(* Logix 5000 project; controller NSH_PLC2 vendor 1 type 14 code 167 rev 32.14; software revision 32.03; part 3 of 6 *)
(* tags used below, declared in another part *)
   AOI_MCC2_15J_ToPLC1 : E300ToMotor;
   AOI_MCC2_15L_ToPLC1 : E300ToMotor;
   AOI_MCC2_16A_ToPLC1 : E300ToMotor;
   AOI_MCC2_16C_ToPLC1 : E300ToMotor;
   AOI_MCC2_16E_ToPLC1 : E300ToMotor;
   AOI_MCC2_16G_ToPLC1 : E300ToMotor;
   AOI_MCC2_16J_ToPLC1 : E300ToMotor;
   AOI_MCC2_16L_ToPLC1 : E300ToMotor;
   AOI_MCC2_17A_ToPLC1 : E300ToMotor;
   AOI_MCC2_17C_ToPLC1 : E300ToMotor;
   AOI_MCC2_17E_ToPLC1 : E300ToMotor;
   AOI_MCC2_17G_ToPLC1 : E300ToMotor;
   AOI_MCC2_17J_ToPLC1 : E300ToMotor;
   AOI_MCC2_18A_ToPLC1 : E300ToMotor;
   AOI_MCC2_18C_ToPLC1 : E300ToMotor;
   AOI_MCC2_18E_ToPLC1 : E300ToMotor;
   AOI_MCC2_18G_ToPLC1 : E300ToMotor;
   AOI_MCC2_18J_ToPLC1 : E300ToMotor;
   AOI_MCC2_18L_ToPLC1 : E300ToMotor;
   AOI_MCC2_19A_ToPLC1 : E300ToMotor;
   AOI_MCC2_19C_ToPLC1 : E300ToMotor;
   AOI_MCC2_19E_ToPLC1 : E300ToMotor;
   AOI_MCC2_19G_ToPLC1 : E300ToMotor;
   AOI_MCC2_19J_ToPLC1 : E300ToMotor;
   AOI_MCC2_19L_ToPLC1 : E300ToMotor;
   AOI_MCC2_20C_ToPLC1 : E300ToMotor;
   AOI_MCC2_20E_ToPLC1 : E300ToMotor;
   AOI_MCC2_20G_ToPLC1 : E300ToMotor;
   AOI_MCC2_20J_ToPLC1 : E300ToMotor;
   AOI_MCC2_21A_ToPLC1 : E300ToMotor;
   AOI_MCC2_21C_ToPLC1 : E300ToMotor;
   AOI_MCC2_21E_ToPLC1 : E300ToMotor;
   AOI_MCC2_21G_ToPLC1 : PF525ToMotor;
   AOI_MCC2_21K_ToPLC1 : PF525ToMotor;
   AOI_MCC3_10A_ToPLC1 : E300ToMotor;
   AOI_MCC3_10D_ToPLC1 : E300ToMotor;
   AOI_MCC3_10G_ToPLC1 : E300ToMotor;
   AOI_MCC3_2A_ToPLC1 : PF525ToMotor;
   AOI_MCC3_2D_ToPLC1 : PF525ToMotor;
   AOI_MCC3_2G_ToPLC1 : PF525ToMotor;
   AOI_MCC3_2K_ToPLC1 : PF525ToMotor;
   AOI_MCC3_3A_ToPLC1 : PF525ToMotor;
   AOI_MCC3_3D_ToPLC1 : PF525ToMotor;
   AOI_MCC3_3G_ToPLC1 : PF525ToMotor;
   AOI_MCC3_3K_ToPLC1 : PF525ToMotor;
   AOI_MCC3_4A_ToPLC1 : PF525ToMotor;
   AOI_MCC3_4D_ToPLC1 : PF525ToMotor;
   AOI_MCC3_4G_ToPLC1 : PF525ToMotor;
   AOI_MCC3_4K_ToPLC1 : PF525ToMotor;
   AOI_MCC3_5A_ToPLC1 : PF525ToMotor;
   AOI_MCC3_5D_ToPLC1 : PF525ToMotor;
   AOI_MCC3_5G_ToPLC1 : PF525ToMotor;
   AOI_MCC3_5K_ToPLC1 : PF525ToMotor;
   AOI_MCC3_6A_ToPLC1 : PF525ToMotor;
   AOI_MCC3_6D_ToPLC1 : PF525ToMotor;
   AOI_MCC3_6G_ToPLC1 : E300ToMotor;
   AOI_MCC3_6J_ToPLC1 : E300ToMotor;
   AOI_MCC3_7A_ToPLC1 : E300ToMotor;
   AOI_MCC3_7C_ToPLC1 : E300ToMotor;
   AOI_MCC3_7E_ToPLC1 : E300ToMotor;
   AOI_MCC3_7G_ToPLC1 : PF525ToMotor;
   AOI_MCC3_7K_ToPLC1 : PF525ToMotor;
   AOI_MCC3_8A_ToPLC1 : E300ToMotor;
   AOI_MCC3_8D_ToPLC1 : PF525ToMotor;
   AOI_MCC3_8H_ToPLC1 : E300ToMotor;
   AOI_MCC3_8K_ToPLC1 : PF525ToMotor;
   AOI_MCC3_9A_ToPLC1 : E300ToMotor;
   AOI_MCC3_9C_ToPLC1 : E300ToMotor;
   AOI_MCC3_9E_ToPLC1 : E300ToMotor;
   AOI_MCC3_9G_ToPLC1 : E300ToMotor;
   AOI_MCC3_9J_ToPLC1 : E300ToMotor;
   AOI_MCC3_9L_ToPLC1 : E300ToMotor;
   Const_4000_Hex : INT;   // Constant #16:4000, Entry Status Communicating
   GSV_EntryStatus : INT;   // GSV Entry Status, shold be #16:4000
   MCC2_15J_CommsOK : BOOL;   // Communications with AOP OK
   MCC2_15L_CommsOK : BOOL;   // Communications with AOP OK
   MCC2_16A_CommsOK : BOOL;   // Communications with AOP OK
   MCC2_16C_CommsOK : BOOL;   // Communications with AOP OK
   MCC2_16E_CommsOK : BOOL;   // Communications with AOP OK
   MCC2_16G_CommsOK : BOOL;   // Communications with AOP OK
   MCC2_16J_CommsOK : BOOL;   // Communications with AOP OK
   MCC2_16L_CommsOK : BOOL;   // Communications with AOP OK
   MCC2_17A_CommsOK : BOOL;   // Communications with AOP OK
   MCC2_17C_CommsOK : BOOL;   // Communications with AOP OK
   MCC2_17E_CommsOK : BOOL;   // Communications with AOP OK
   MCC2_17G_CommsOK : BOOL;   // Communications with AOP OK
   MCC2_17J_CommsOK : BOOL;   // Communications with AOP OK
   MCC2_18A_CommsOK : BOOL;   // Communications with AOP OK
   MCC2_18C_CommsOK : BOOL;   // Communications with AOP OK
   MCC2_18E_CommsOK : BOOL;   // Communications with AOP OK
   MCC2_18G_CommsOK : BOOL;   // Communications with AOP OK
   MCC2_18J_CommsOK : BOOL;   // Communications with AOP OK
   MCC2_18L_CommsOK : BOOL;   // Communications with AOP OK
   MCC2_19A_CommsOK : BOOL;   // Communications with AOP OK
   MCC2_19C_CommsOK : BOOL;   // Communications with AOP OK
   MCC2_19E_CommsOK : BOOL;   // Communications with AOP OK
   MCC2_19G_CommsOK : BOOL;   // Communications with AOP OK
   MCC2_19J_CommsOK : BOOL;   // Communications with AOP OK
   MCC2_19L_CommsOK : BOOL;   // Communications with AOP OK
   MCC2_20C_CommsOK : BOOL;   // Communications with AOP OK
   MCC2_20E_CommsOK : BOOL;   // Communications with AOP OK
   MCC2_20G_CommsOK : BOOL;   // Communications with AOP OK
   MCC2_20J_CommsOK : BOOL;   // Communications with AOP OK
   MCC2_21A_CommsOK : BOOL;   // Communications with AOP OK
   MCC2_21C_CommsOK : BOOL;   // Communications with AOP OK
   MCC2_21E_CommsOK : BOOL;   // Communications with AOP OK
   MCC2_21G_CommsOK : BOOL;   // Communications with AOP OK
   MCC2_21K_CommsOK : BOOL;   // Communications with AOP OK
   MCC3_10A_CommsOK : BOOL;   // Communications with AOP OK
   MCC3_10D_CommsOK : BOOL;   // Communications with AOP OK
   MCC3_10G_CommsOK : BOOL;   // Communications with AOP OK
   MCC3_2A_CommsOK : BOOL;   // Communications with AOP OK
   MCC3_2D_CommsOK : BOOL;   // Communications with AOP OK
   MCC3_2G_CommsOK : BOOL;   // Communications with AOP OK
   MCC3_2K_CommsOK : BOOL;   // Communications with AOP OK
   MCC3_3A_CommsOK : BOOL;   // Communications with AOP OK
   MCC3_3D_CommsOK : BOOL;   // Communications with AOP OK
   MCC3_3G_CommsOK : BOOL;   // Communications with AOP OK
   MCC3_3K_CommsOK : BOOL;   // Communications with AOP OK
   MCC3_4A_CommsOK : BOOL;   // Communications with AOP OK
   MCC3_4D_CommsOK : BOOL;   // Communications with AOP OK
   MCC3_4G_CommsOK : BOOL;   // Communications with AOP OK
   MCC3_4K_CommsOK : BOOL;   // Communications with AOP OK
   MCC3_5A_CommsOK : BOOL;   // Communications with AOP OK
   MCC3_5D_CommsOK : BOOL;   // Communications with AOP OK
   MCC3_5G_CommsOK : BOOL;   // Communications with AOP OK
   MCC3_5K_CommsOK : BOOL;   // Communications with AOP OK
   MCC3_6A_CommsOK : BOOL;   // Communications with AOP OK
   MCC3_6D_CommsOK : BOOL;   // Communications with AOP OK
   MCC3_6G_CommsOK : BOOL;   // Communications with AOP OK
   MCC3_6J_CommsOK : BOOL;   // Communications with AOP OK
   MCC3_7A_CommsOK : BOOL;   // Communications with AOP OK
   MCC3_7C_CommsOK : BOOL;   // Communications with AOP OK
   MCC3_7E_CommsOK : BOOL;   // Communications with AOP OK
   MCC3_7G_CommsOK : BOOL;   // Communications with AOP OK
   MCC3_7K_CommsOK : BOOL;   // Communications with AOP OK
   MCC3_8A_CommsOK : BOOL;   // Communications with AOP OK
   MCC3_8D_CommsOK : BOOL;   // Communications with AOP OK
   MCC3_8H_CommsOK : BOOL;   // Communications with AOP OK
   MCC3_8K_CommsOK : BOOL;   // Communications with AOP OK
   MCC3_9A_CommsOK : BOOL;   // Communications with AOP OK
   MCC3_9C_CommsOK : BOOL;   // Communications with AOP OK
   MCC3_9E_CommsOK : BOOL;   // Communications with AOP OK
   MCC3_9G_CommsOK : BOOL;   // Communications with AOP OK
   MCC3_9J_CommsOK : BOOL;   // Communications with AOP OK
   MCC3_9L_CommsOK : BOOL;   // Communications with AOP OK
   MotorsStatusTag : MotorsStatusUDT;   // Only Instance of UDT
(* MainProgram, continued *)

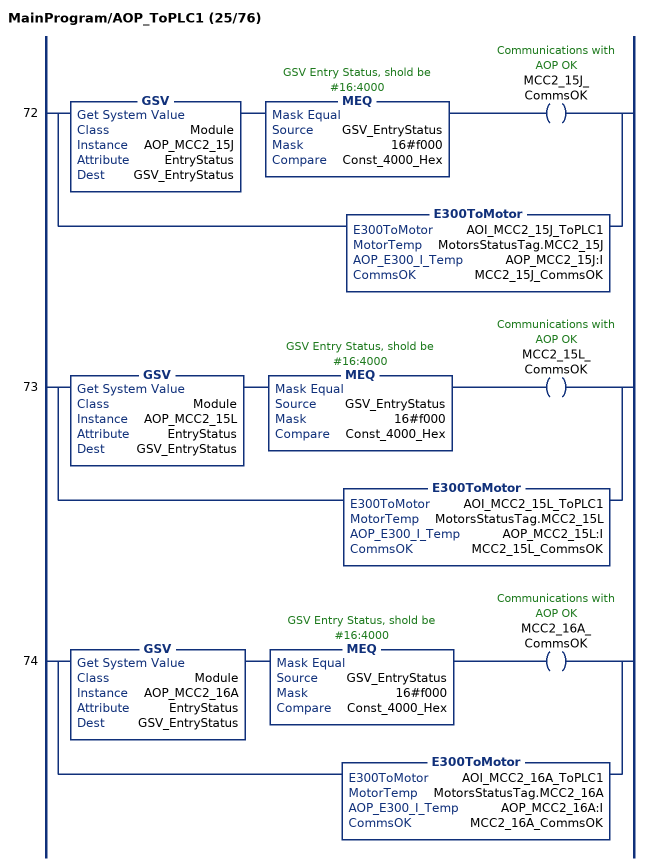
   [picture p31: MainProgram/AOP_ToPLC1 rungs 72-74]
   72: [GSV(Module,AOP_MCC2_15J,EntryStatus,GSV_EntryStatus) MEQ(GSV_EntryStatus,16#f000,Const_4000_Hex) OTE(MCC2_15J_CommsOK) ,E300ToMotor(AOI_MCC2_15J_ToPLC1,MotorsStatusTag.MCC2_15J,AOP_MCC2_15J:I,MCC2_15J_CommsOK) ];
   73: [GSV(Module,AOP_MCC2_15L,EntryStatus,GSV_EntryStatus) MEQ(GSV_EntryStatus,16#f000,Const_4000_Hex) OTE(MCC2_15L_CommsOK) ,E300ToMotor(AOI_MCC2_15L_ToPLC1,MotorsStatusTag.MCC2_15L,AOP_MCC2_15L:I,MCC2_15L_CommsOK) ];
   74: [GSV(Module,AOP_MCC2_16A,EntryStatus,GSV_EntryStatus) MEQ(GSV_EntryStatus,16#f000,Const_4000_Hex) OTE(MCC2_16A_CommsOK) ,E300ToMotor(AOI_MCC2_16A_ToPLC1,MotorsStatusTag.MCC2_16A,AOP_MCC2_16A:I,MCC2_16A_CommsOK) ];
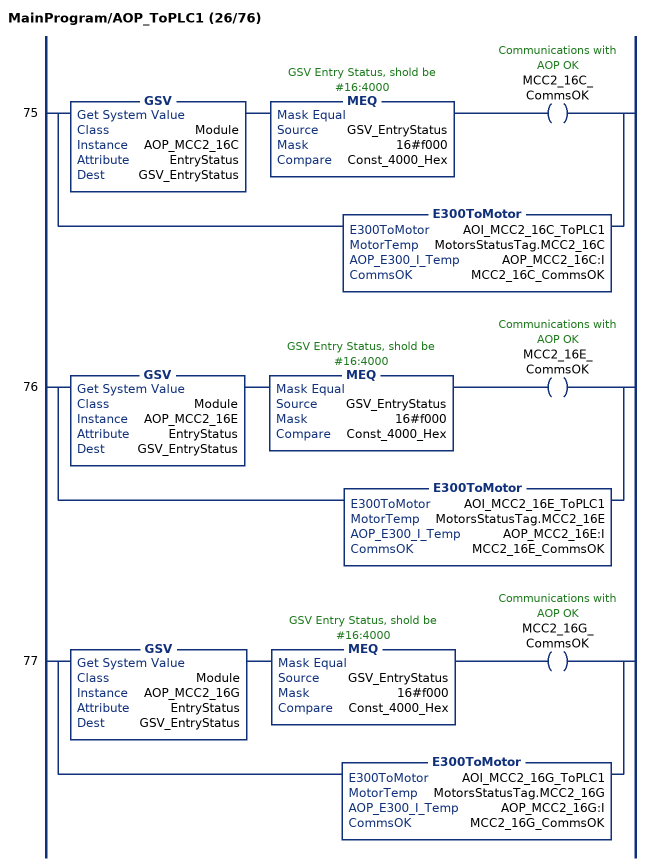
   75: [GSV(Module,AOP_MCC2_16C,EntryStatus,GSV_EntryStatus) MEQ(GSV_EntryStatus,16#f000,Const_4000_Hex) OTE(MCC2_16C_CommsOK) ,E300ToMotor(AOI_MCC2_16C_ToPLC1,MotorsStatusTag.MCC2_16C,AOP_MCC2_16C:I,MCC2_16C_CommsOK) ];
   76: [GSV(Module,AOP_MCC2_16E,EntryStatus,GSV_EntryStatus) MEQ(GSV_EntryStatus,16#f000,Const_4000_Hex) OTE(MCC2_16E_CommsOK) ,E300ToMotor(AOI_MCC2_16E_ToPLC1,MotorsStatusTag.MCC2_16E,AOP_MCC2_16E:I,MCC2_16E_CommsOK) ];
   77: [GSV(Module,AOP_MCC2_16G,EntryStatus,GSV_EntryStatus) MEQ(GSV_EntryStatus,16#f000,Const_4000_Hex) OTE(MCC2_16G_CommsOK) ,E300ToMotor(AOI_MCC2_16G_ToPLC1,MotorsStatusTag.MCC2_16G,AOP_MCC2_16G:I,MCC2_16G_CommsOK) ];
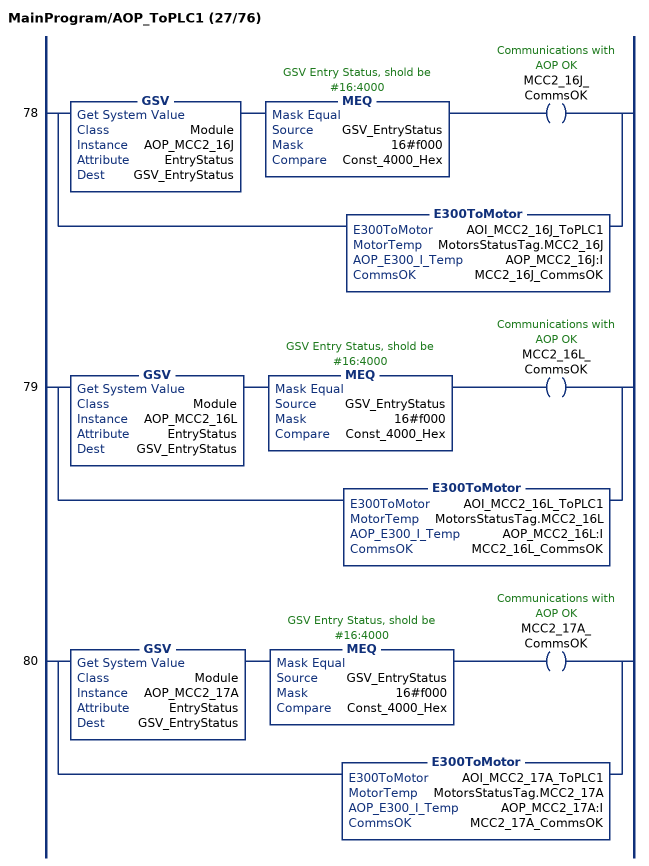
   78: [GSV(Module,AOP_MCC2_16J,EntryStatus,GSV_EntryStatus) MEQ(GSV_EntryStatus,16#f000,Const_4000_Hex) OTE(MCC2_16J_CommsOK) ,E300ToMotor(AOI_MCC2_16J_ToPLC1,MotorsStatusTag.MCC2_16J,AOP_MCC2_16J:I,MCC2_16J_CommsOK) ];
   79: [GSV(Module,AOP_MCC2_16L,EntryStatus,GSV_EntryStatus) MEQ(GSV_EntryStatus,16#f000,Const_4000_Hex) OTE(MCC2_16L_CommsOK) ,E300ToMotor(AOI_MCC2_16L_ToPLC1,MotorsStatusTag.MCC2_16L,AOP_MCC2_16L:I,MCC2_16L_CommsOK) ];
   80: [GSV(Module,AOP_MCC2_17A,EntryStatus,GSV_EntryStatus) MEQ(GSV_EntryStatus,16#f000,Const_4000_Hex) OTE(MCC2_17A_CommsOK) ,E300ToMotor(AOI_MCC2_17A_ToPLC1,MotorsStatusTag.MCC2_17A,AOP_MCC2_17A:I,MCC2_17A_CommsOK) ];
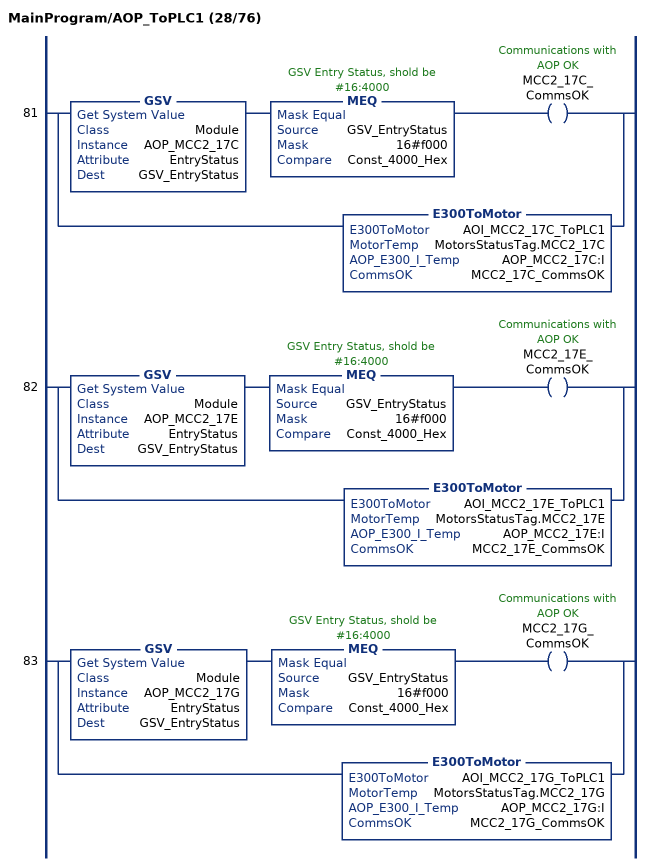
   81: [GSV(Module,AOP_MCC2_17C,EntryStatus,GSV_EntryStatus) MEQ(GSV_EntryStatus,16#f000,Const_4000_Hex) OTE(MCC2_17C_CommsOK) ,E300ToMotor(AOI_MCC2_17C_ToPLC1,MotorsStatusTag.MCC2_17C,AOP_MCC2_17C:I,MCC2_17C_CommsOK) ];
   82: [GSV(Module,AOP_MCC2_17E,EntryStatus,GSV_EntryStatus) MEQ(GSV_EntryStatus,16#f000,Const_4000_Hex) OTE(MCC2_17E_CommsOK) ,E300ToMotor(AOI_MCC2_17E_ToPLC1,MotorsStatusTag.MCC2_17E,AOP_MCC2_17E:I,MCC2_17E_CommsOK) ];
   83: [GSV(Module,AOP_MCC2_17G,EntryStatus,GSV_EntryStatus) MEQ(GSV_EntryStatus,16#f000,Const_4000_Hex) OTE(MCC2_17G_CommsOK) ,E300ToMotor(AOI_MCC2_17G_ToPLC1,MotorsStatusTag.MCC2_17G,AOP_MCC2_17G:I,MCC2_17G_CommsOK) ];
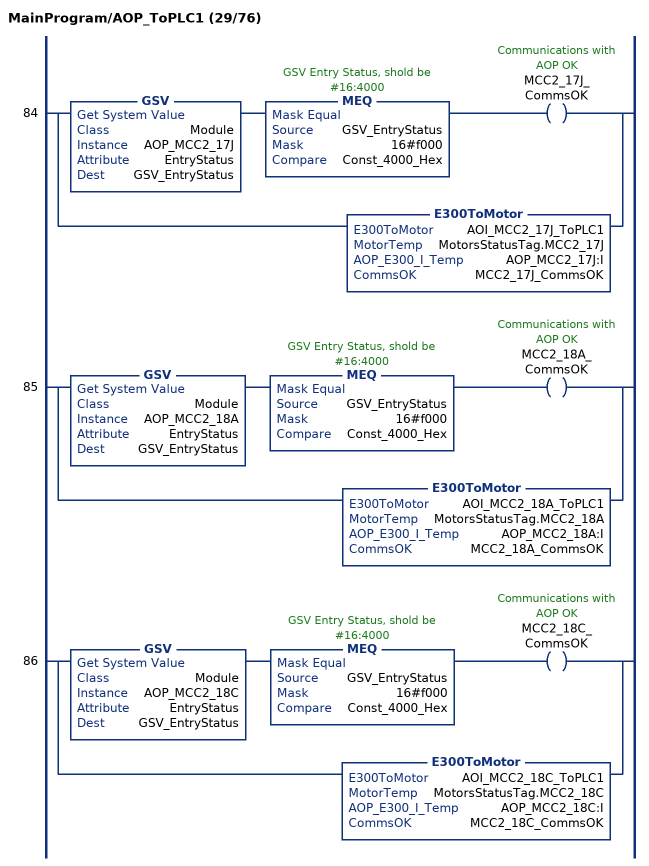
   84: [GSV(Module,AOP_MCC2_17J,EntryStatus,GSV_EntryStatus) MEQ(GSV_EntryStatus,16#f000,Const_4000_Hex) OTE(MCC2_17J_CommsOK) ,E300ToMotor(AOI_MCC2_17J_ToPLC1,MotorsStatusTag.MCC2_17J,AOP_MCC2_17J:I,MCC2_17J_CommsOK) ];
   85: [GSV(Module,AOP_MCC2_18A,EntryStatus,GSV_EntryStatus) MEQ(GSV_EntryStatus,16#f000,Const_4000_Hex) OTE(MCC2_18A_CommsOK) ,E300ToMotor(AOI_MCC2_18A_ToPLC1,MotorsStatusTag.MCC2_18A,AOP_MCC2_18A:I,MCC2_18A_CommsOK) ];
   86: [GSV(Module,AOP_MCC2_18C,EntryStatus,GSV_EntryStatus) MEQ(GSV_EntryStatus,16#f000,Const_4000_Hex) OTE(MCC2_18C_CommsOK) ,E300ToMotor(AOI_MCC2_18C_ToPLC1,MotorsStatusTag.MCC2_18C,AOP_MCC2_18C:I,MCC2_18C_CommsOK) ];
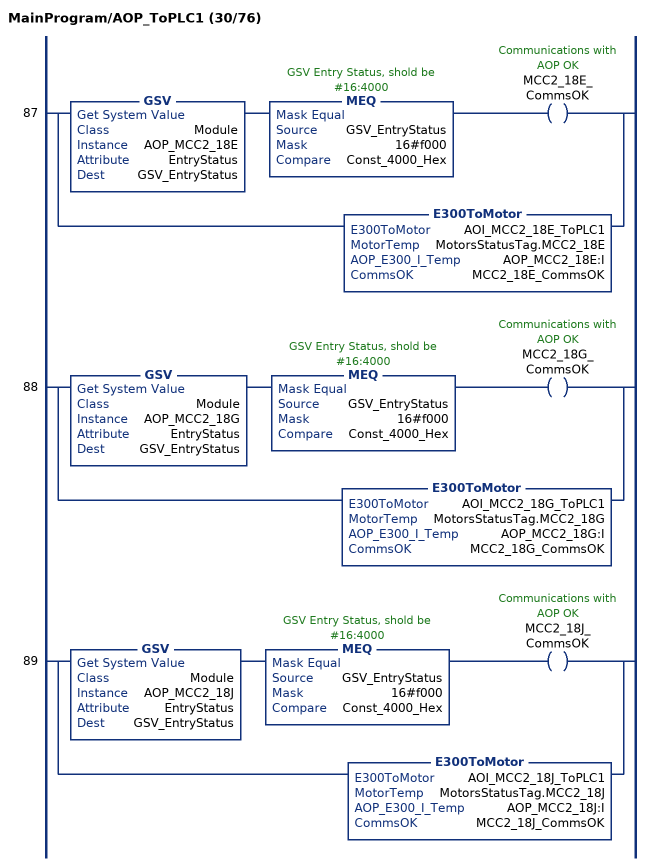
   87: [GSV(Module,AOP_MCC2_18E,EntryStatus,GSV_EntryStatus) MEQ(GSV_EntryStatus,16#f000,Const_4000_Hex) OTE(MCC2_18E_CommsOK) ,E300ToMotor(AOI_MCC2_18E_ToPLC1,MotorsStatusTag.MCC2_18E,AOP_MCC2_18E:I,MCC2_18E_CommsOK) ];
   88: [GSV(Module,AOP_MCC2_18G,EntryStatus,GSV_EntryStatus) MEQ(GSV_EntryStatus,16#f000,Const_4000_Hex) OTE(MCC2_18G_CommsOK) ,E300ToMotor(AOI_MCC2_18G_ToPLC1,MotorsStatusTag.MCC2_18G,AOP_MCC2_18G:I,MCC2_18G_CommsOK) ];
   89: [GSV(Module,AOP_MCC2_18J,EntryStatus,GSV_EntryStatus) MEQ(GSV_EntryStatus,16#f000,Const_4000_Hex) OTE(MCC2_18J_CommsOK) ,E300ToMotor(AOI_MCC2_18J_ToPLC1,MotorsStatusTag.MCC2_18J,AOP_MCC2_18J:I,MCC2_18J_CommsOK) ];
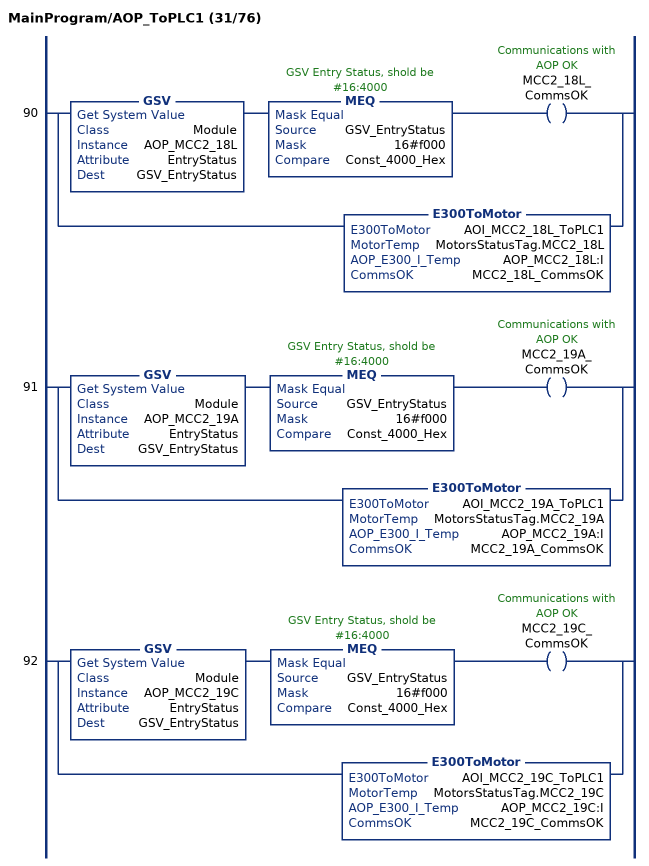
   90: [GSV(Module,AOP_MCC2_18L,EntryStatus,GSV_EntryStatus) MEQ(GSV_EntryStatus,16#f000,Const_4000_Hex) OTE(MCC2_18L_CommsOK) ,E300ToMotor(AOI_MCC2_18L_ToPLC1,MotorsStatusTag.MCC2_18L,AOP_MCC2_18L:I,MCC2_18L_CommsOK) ];
   91: [GSV(Module,AOP_MCC2_19A,EntryStatus,GSV_EntryStatus) MEQ(GSV_EntryStatus,16#f000,Const_4000_Hex) OTE(MCC2_19A_CommsOK) ,E300ToMotor(AOI_MCC2_19A_ToPLC1,MotorsStatusTag.MCC2_19A,AOP_MCC2_19A:I,MCC2_19A_CommsOK) ];
   92: [GSV(Module,AOP_MCC2_19C,EntryStatus,GSV_EntryStatus) MEQ(GSV_EntryStatus,16#f000,Const_4000_Hex) OTE(MCC2_19C_CommsOK) ,E300ToMotor(AOI_MCC2_19C_ToPLC1,MotorsStatusTag.MCC2_19C,AOP_MCC2_19C:I,MCC2_19C_CommsOK) ];
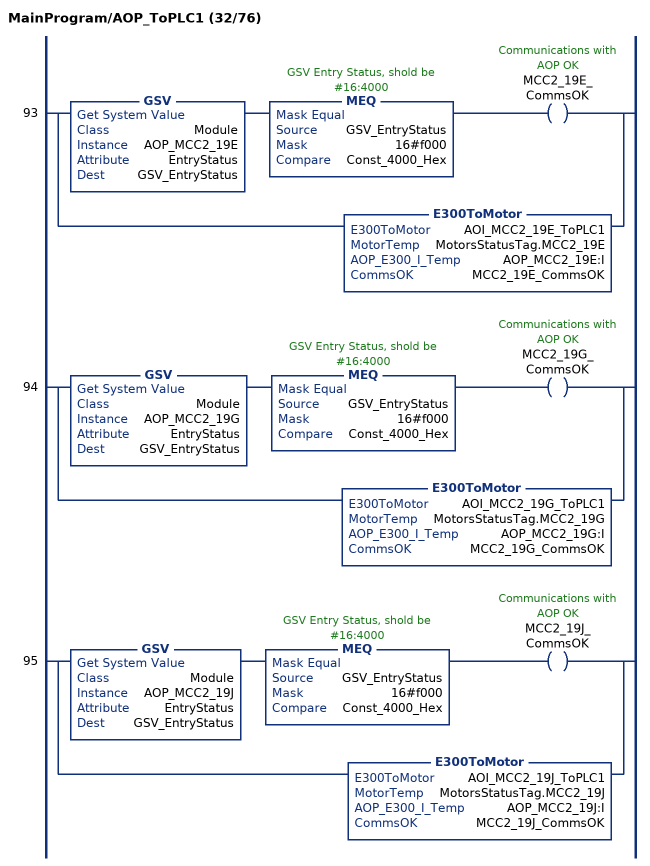
   93: [GSV(Module,AOP_MCC2_19E,EntryStatus,GSV_EntryStatus) MEQ(GSV_EntryStatus,16#f000,Const_4000_Hex) OTE(MCC2_19E_CommsOK) ,E300ToMotor(AOI_MCC2_19E_ToPLC1,MotorsStatusTag.MCC2_19E,AOP_MCC2_19E:I,MCC2_19E_CommsOK) ];
   94: [GSV(Module,AOP_MCC2_19G,EntryStatus,GSV_EntryStatus) MEQ(GSV_EntryStatus,16#f000,Const_4000_Hex) OTE(MCC2_19G_CommsOK) ,E300ToMotor(AOI_MCC2_19G_ToPLC1,MotorsStatusTag.MCC2_19G,AOP_MCC2_19G:I,MCC2_19G_CommsOK) ];
   95: [GSV(Module,AOP_MCC2_19J,EntryStatus,GSV_EntryStatus) MEQ(GSV_EntryStatus,16#f000,Const_4000_Hex) OTE(MCC2_19J_CommsOK) ,E300ToMotor(AOI_MCC2_19J_ToPLC1,MotorsStatusTag.MCC2_19J,AOP_MCC2_19J:I,MCC2_19J_CommsOK) ];
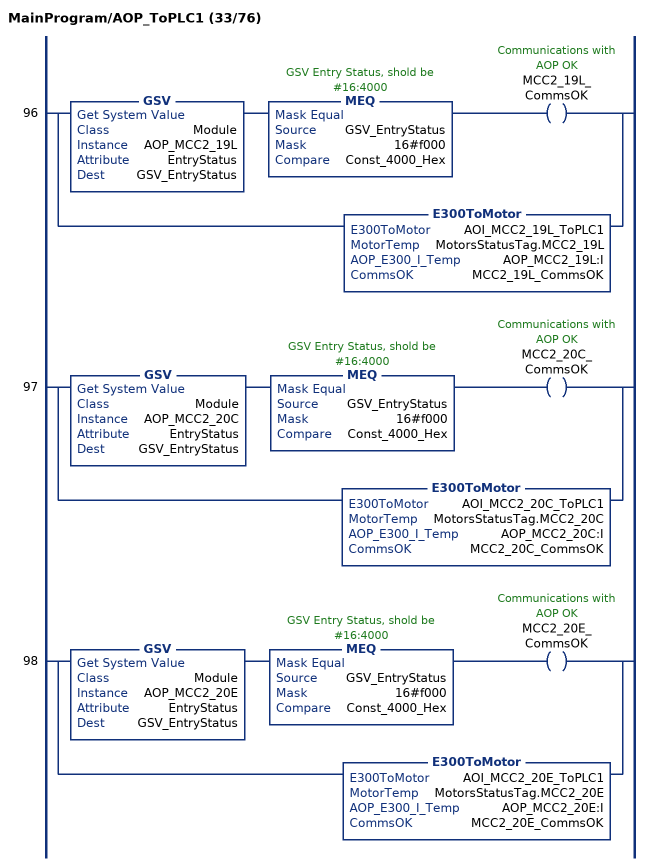
   96: [GSV(Module,AOP_MCC2_19L,EntryStatus,GSV_EntryStatus) MEQ(GSV_EntryStatus,16#f000,Const_4000_Hex) OTE(MCC2_19L_CommsOK) ,E300ToMotor(AOI_MCC2_19L_ToPLC1,MotorsStatusTag.MCC2_19L,AOP_MCC2_19L:I,MCC2_19L_CommsOK) ];
   97: [GSV(Module,AOP_MCC2_20C,EntryStatus,GSV_EntryStatus) MEQ(GSV_EntryStatus,16#f000,Const_4000_Hex) OTE(MCC2_20C_CommsOK) ,E300ToMotor(AOI_MCC2_20C_ToPLC1,MotorsStatusTag.MCC2_20C,AOP_MCC2_20C:I,MCC2_20C_CommsOK) ];
   98: [GSV(Module,AOP_MCC2_20E,EntryStatus,GSV_EntryStatus) MEQ(GSV_EntryStatus,16#f000,Const_4000_Hex) OTE(MCC2_20E_CommsOK) ,E300ToMotor(AOI_MCC2_20E_ToPLC1,MotorsStatusTag.MCC2_20E,AOP_MCC2_20E:I,MCC2_20E_CommsOK) ];
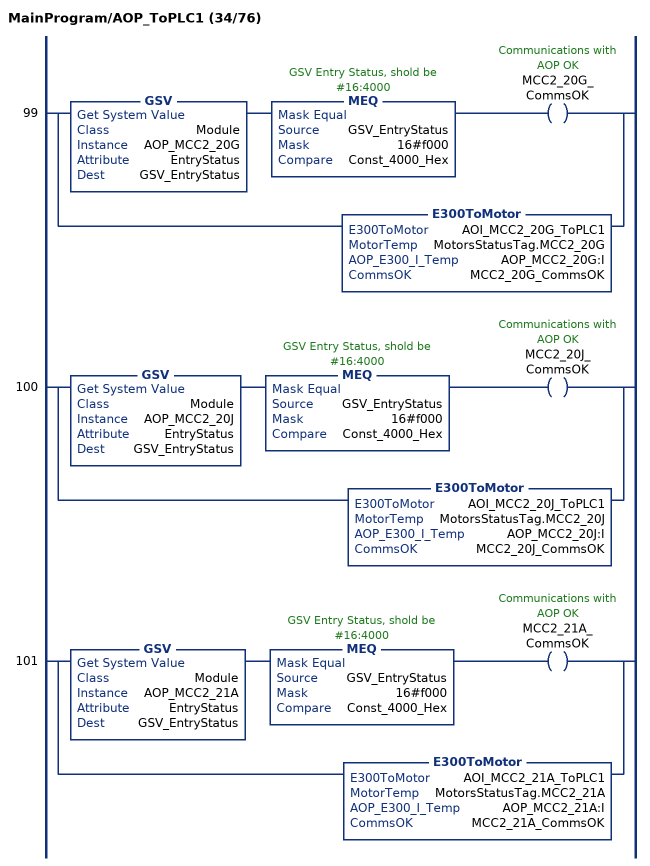
   99: [GSV(Module,AOP_MCC2_20G,EntryStatus,GSV_EntryStatus) MEQ(GSV_EntryStatus,16#f000,Const_4000_Hex) OTE(MCC2_20G_CommsOK) ,E300ToMotor(AOI_MCC2_20G_ToPLC1,MotorsStatusTag.MCC2_20G,AOP_MCC2_20G:I,MCC2_20G_CommsOK) ];
   100: [GSV(Module,AOP_MCC2_20J,EntryStatus,GSV_EntryStatus) MEQ(GSV_EntryStatus,16#f000,Const_4000_Hex) OTE(MCC2_20J_CommsOK) ,E300ToMotor(AOI_MCC2_20J_ToPLC1,MotorsStatusTag.MCC2_20J,AOP_MCC2_20J:I,MCC2_20J_CommsOK) ];
   101: [GSV(Module,AOP_MCC2_21A,EntryStatus,GSV_EntryStatus) MEQ(GSV_EntryStatus,16#f000,Const_4000_Hex) OTE(MCC2_21A_CommsOK) ,E300ToMotor(AOI_MCC2_21A_ToPLC1,MotorsStatusTag.MCC2_21A,AOP_MCC2_21A:I,MCC2_21A_CommsOK) ];
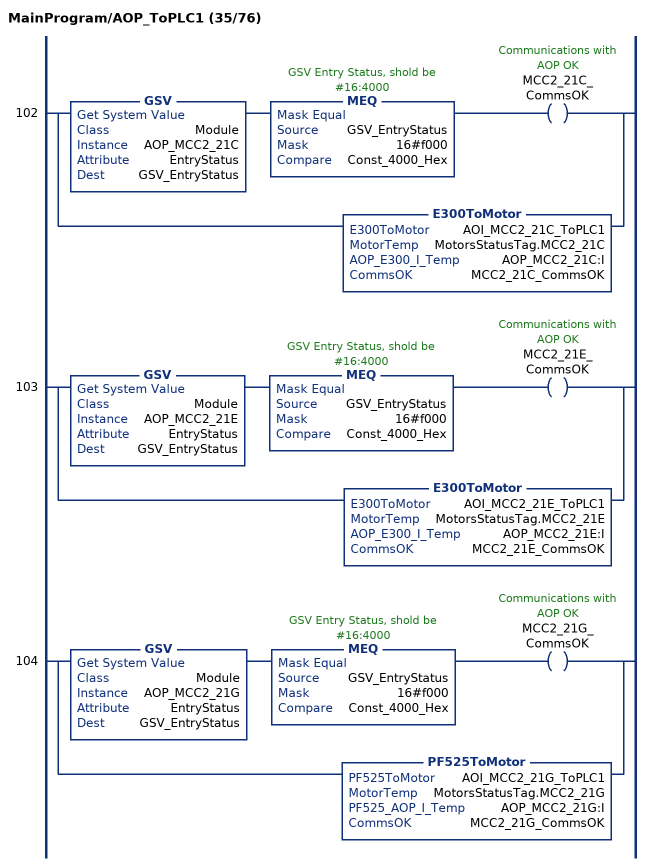
   102: [GSV(Module,AOP_MCC2_21C,EntryStatus,GSV_EntryStatus) MEQ(GSV_EntryStatus,16#f000,Const_4000_Hex) OTE(MCC2_21C_CommsOK) ,E300ToMotor(AOI_MCC2_21C_ToPLC1,MotorsStatusTag.MCC2_21C,AOP_MCC2_21C:I,MCC2_21C_CommsOK) ];
   103: [GSV(Module,AOP_MCC2_21E,EntryStatus,GSV_EntryStatus) MEQ(GSV_EntryStatus,16#f000,Const_4000_Hex) OTE(MCC2_21E_CommsOK) ,E300ToMotor(AOI_MCC2_21E_ToPLC1,MotorsStatusTag.MCC2_21E,AOP_MCC2_21E:I,MCC2_21E_CommsOK) ];
   104: [GSV(Module,AOP_MCC2_21G,EntryStatus,GSV_EntryStatus) MEQ(GSV_EntryStatus,16#f000,Const_4000_Hex) OTE(MCC2_21G_CommsOK) ,PF525ToMotor(AOI_MCC2_21G_ToPLC1,MotorsStatusTag.MCC2_21G,AOP_MCC2_21G:I,MCC2_21G_CommsOK) ];
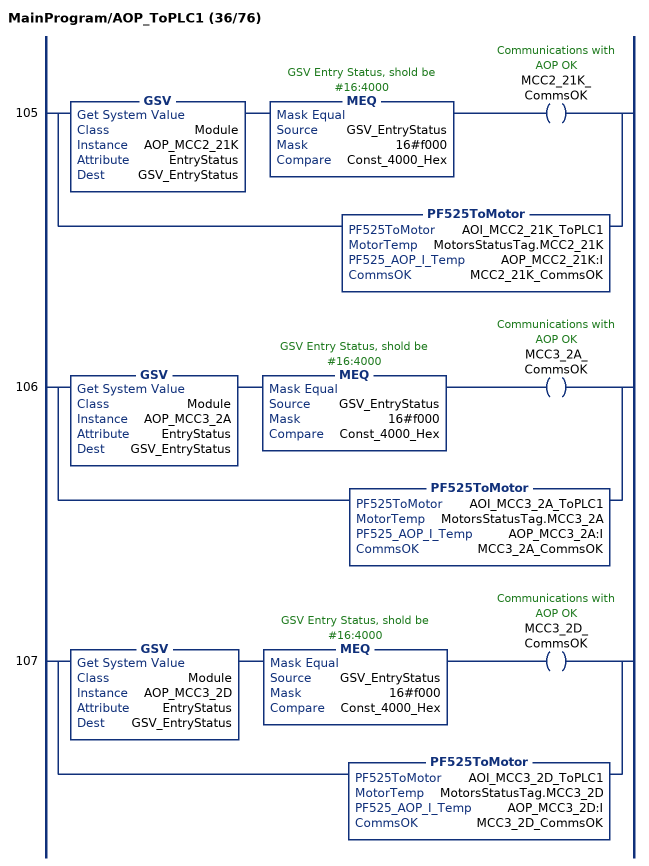
   105: [GSV(Module,AOP_MCC2_21K,EntryStatus,GSV_EntryStatus) MEQ(GSV_EntryStatus,16#f000,Const_4000_Hex) OTE(MCC2_21K_CommsOK) ,PF525ToMotor(AOI_MCC2_21K_ToPLC1,MotorsStatusTag.MCC2_21K,AOP_MCC2_21K:I,MCC2_21K_CommsOK) ];
   106: [GSV(Module,AOP_MCC3_2A,EntryStatus,GSV_EntryStatus) MEQ(GSV_EntryStatus,16#f000,Const_4000_Hex) OTE(MCC3_2A_CommsOK) ,PF525ToMotor(AOI_MCC3_2A_ToPLC1,MotorsStatusTag.MCC3_2A,AOP_MCC3_2A:I,MCC3_2A_CommsOK) ];
   107: [GSV(Module,AOP_MCC3_2D,EntryStatus,GSV_EntryStatus) MEQ(GSV_EntryStatus,16#f000,Const_4000_Hex) OTE(MCC3_2D_CommsOK) ,PF525ToMotor(AOI_MCC3_2D_ToPLC1,MotorsStatusTag.MCC3_2D,AOP_MCC3_2D:I,MCC3_2D_CommsOK) ];
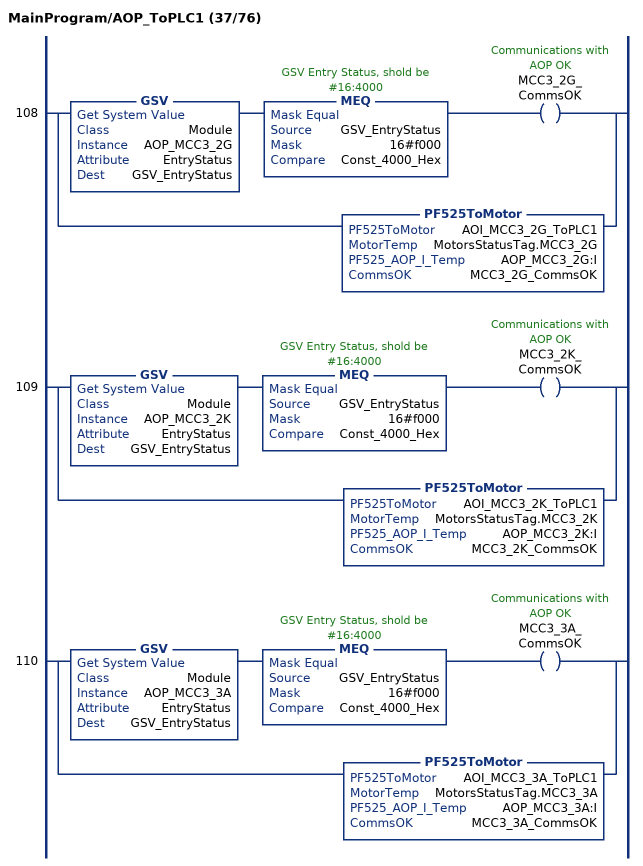
   108: [GSV(Module,AOP_MCC3_2G,EntryStatus,GSV_EntryStatus) MEQ(GSV_EntryStatus,16#f000,Const_4000_Hex) OTE(MCC3_2G_CommsOK) ,PF525ToMotor(AOI_MCC3_2G_ToPLC1,MotorsStatusTag.MCC3_2G,AOP_MCC3_2G:I,MCC3_2G_CommsOK) ];
   109: [GSV(Module,AOP_MCC3_2K,EntryStatus,GSV_EntryStatus) MEQ(GSV_EntryStatus,16#f000,Const_4000_Hex) OTE(MCC3_2K_CommsOK) ,PF525ToMotor(AOI_MCC3_2K_ToPLC1,MotorsStatusTag.MCC3_2K,AOP_MCC3_2K:I,MCC3_2K_CommsOK) ];
   110: [GSV(Module,AOP_MCC3_3A,EntryStatus,GSV_EntryStatus) MEQ(GSV_EntryStatus,16#f000,Const_4000_Hex) OTE(MCC3_3A_CommsOK) ,PF525ToMotor(AOI_MCC3_3A_ToPLC1,MotorsStatusTag.MCC3_3A,AOP_MCC3_3A:I,MCC3_3A_CommsOK) ];
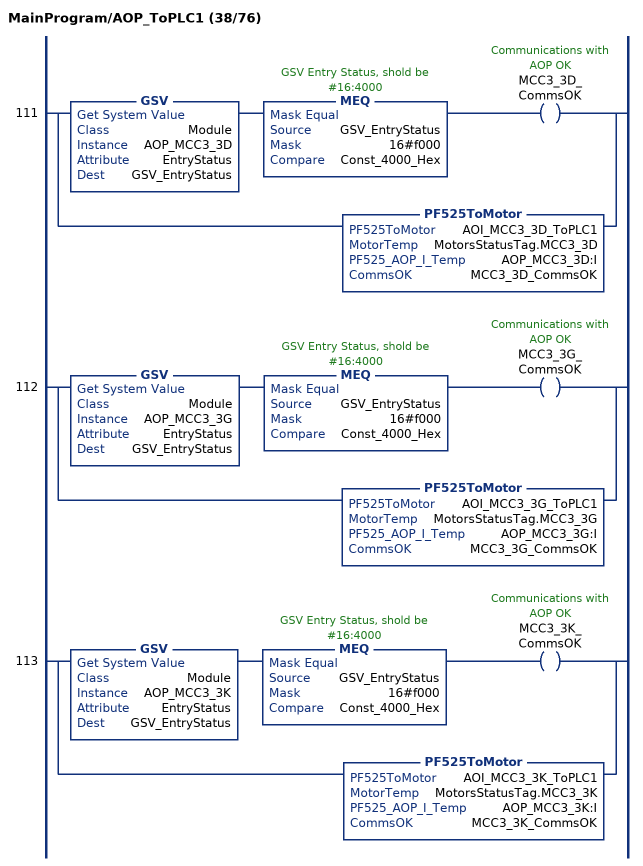
   111: [GSV(Module,AOP_MCC3_3D,EntryStatus,GSV_EntryStatus) MEQ(GSV_EntryStatus,16#f000,Const_4000_Hex) OTE(MCC3_3D_CommsOK) ,PF525ToMotor(AOI_MCC3_3D_ToPLC1,MotorsStatusTag.MCC3_3D,AOP_MCC3_3D:I,MCC3_3D_CommsOK) ];
   112: [GSV(Module,AOP_MCC3_3G,EntryStatus,GSV_EntryStatus) MEQ(GSV_EntryStatus,16#f000,Const_4000_Hex) OTE(MCC3_3G_CommsOK) ,PF525ToMotor(AOI_MCC3_3G_ToPLC1,MotorsStatusTag.MCC3_3G,AOP_MCC3_3G:I,MCC3_3G_CommsOK) ];
   113: [GSV(Module,AOP_MCC3_3K,EntryStatus,GSV_EntryStatus) MEQ(GSV_EntryStatus,16#f000,Const_4000_Hex) OTE(MCC3_3K_CommsOK) ,PF525ToMotor(AOI_MCC3_3K_ToPLC1,MotorsStatusTag.MCC3_3K,AOP_MCC3_3K:I,MCC3_3K_CommsOK) ];
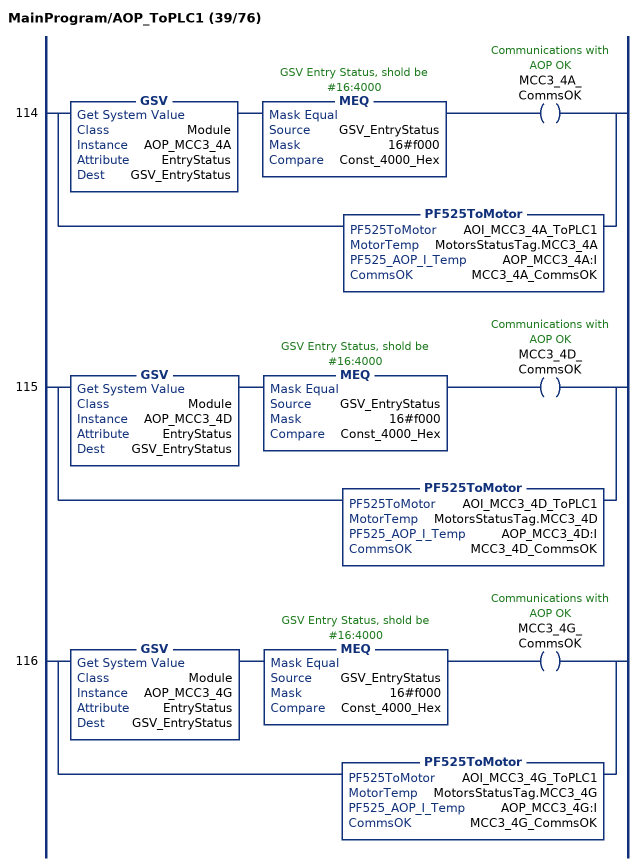
   114: [GSV(Module,AOP_MCC3_4A,EntryStatus,GSV_EntryStatus) MEQ(GSV_EntryStatus,16#f000,Const_4000_Hex) OTE(MCC3_4A_CommsOK) ,PF525ToMotor(AOI_MCC3_4A_ToPLC1,MotorsStatusTag.MCC3_4A,AOP_MCC3_4A:I,MCC3_4A_CommsOK) ];
   115: [GSV(Module,AOP_MCC3_4D,EntryStatus,GSV_EntryStatus) MEQ(GSV_EntryStatus,16#f000,Const_4000_Hex) OTE(MCC3_4D_CommsOK) ,PF525ToMotor(AOI_MCC3_4D_ToPLC1,MotorsStatusTag.MCC3_4D,AOP_MCC3_4D:I,MCC3_4D_CommsOK) ];
   116: [GSV(Module,AOP_MCC3_4G,EntryStatus,GSV_EntryStatus) MEQ(GSV_EntryStatus,16#f000,Const_4000_Hex) OTE(MCC3_4G_CommsOK) ,PF525ToMotor(AOI_MCC3_4G_ToPLC1,MotorsStatusTag.MCC3_4G,AOP_MCC3_4G:I,MCC3_4G_CommsOK) ];
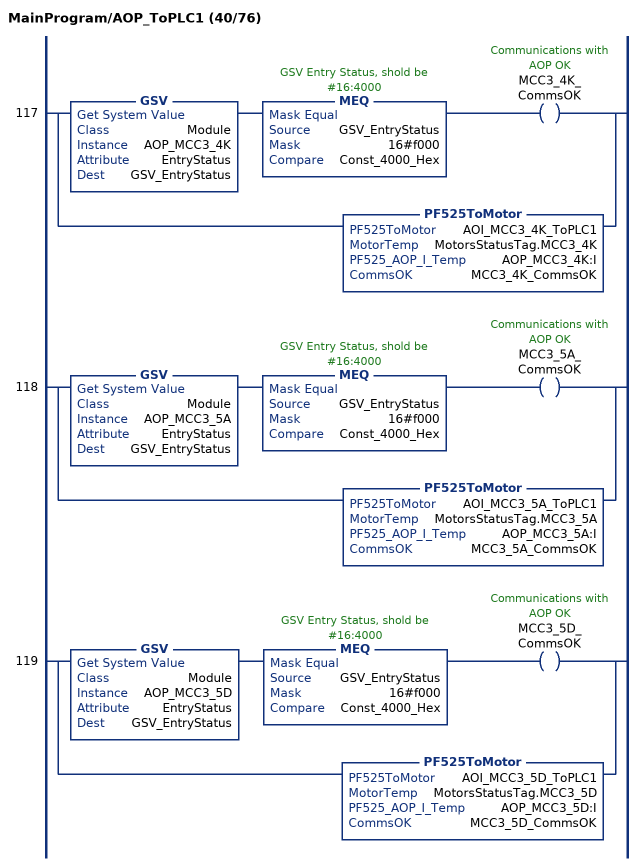
   117: [GSV(Module,AOP_MCC3_4K,EntryStatus,GSV_EntryStatus) MEQ(GSV_EntryStatus,16#f000,Const_4000_Hex) OTE(MCC3_4K_CommsOK) ,PF525ToMotor(AOI_MCC3_4K_ToPLC1,MotorsStatusTag.MCC3_4K,AOP_MCC3_4K:I,MCC3_4K_CommsOK) ];
   118: [GSV(Module,AOP_MCC3_5A,EntryStatus,GSV_EntryStatus) MEQ(GSV_EntryStatus,16#f000,Const_4000_Hex) OTE(MCC3_5A_CommsOK) ,PF525ToMotor(AOI_MCC3_5A_ToPLC1,MotorsStatusTag.MCC3_5A,AOP_MCC3_5A:I,MCC3_5A_CommsOK) ];
   119: [GSV(Module,AOP_MCC3_5D,EntryStatus,GSV_EntryStatus) MEQ(GSV_EntryStatus,16#f000,Const_4000_Hex) OTE(MCC3_5D_CommsOK) ,PF525ToMotor(AOI_MCC3_5D_ToPLC1,MotorsStatusTag.MCC3_5D,AOP_MCC3_5D:I,MCC3_5D_CommsOK) ];
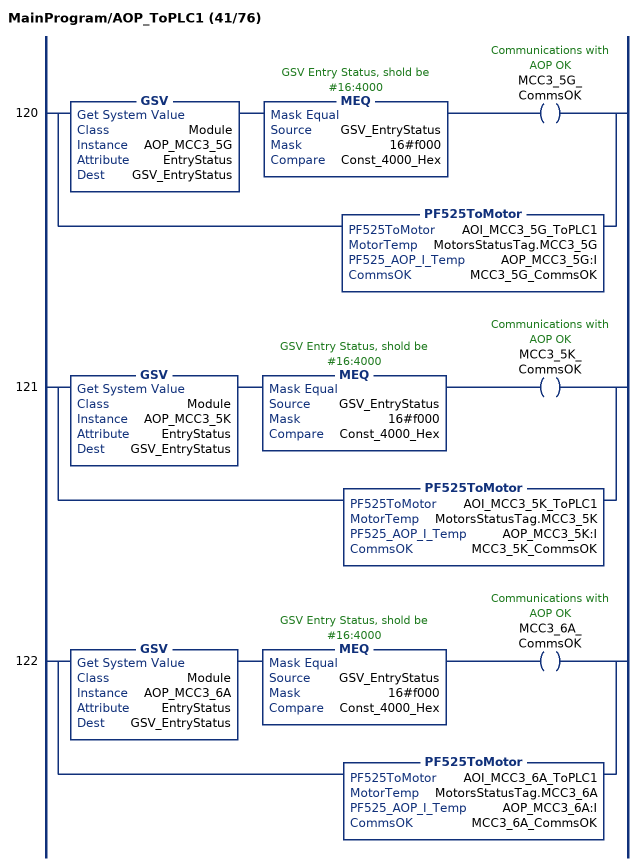
   120: [GSV(Module,AOP_MCC3_5G,EntryStatus,GSV_EntryStatus) MEQ(GSV_EntryStatus,16#f000,Const_4000_Hex) OTE(MCC3_5G_CommsOK) ,PF525ToMotor(AOI_MCC3_5G_ToPLC1,MotorsStatusTag.MCC3_5G,AOP_MCC3_5G:I,MCC3_5G_CommsOK) ];
   121: [GSV(Module,AOP_MCC3_5K,EntryStatus,GSV_EntryStatus) MEQ(GSV_EntryStatus,16#f000,Const_4000_Hex) OTE(MCC3_5K_CommsOK) ,PF525ToMotor(AOI_MCC3_5K_ToPLC1,MotorsStatusTag.MCC3_5K,AOP_MCC3_5K:I,MCC3_5K_CommsOK) ];
   122: [GSV(Module,AOP_MCC3_6A,EntryStatus,GSV_EntryStatus) MEQ(GSV_EntryStatus,16#f000,Const_4000_Hex) OTE(MCC3_6A_CommsOK) ,PF525ToMotor(AOI_MCC3_6A_ToPLC1,MotorsStatusTag.MCC3_6A,AOP_MCC3_6A:I,MCC3_6A_CommsOK) ];
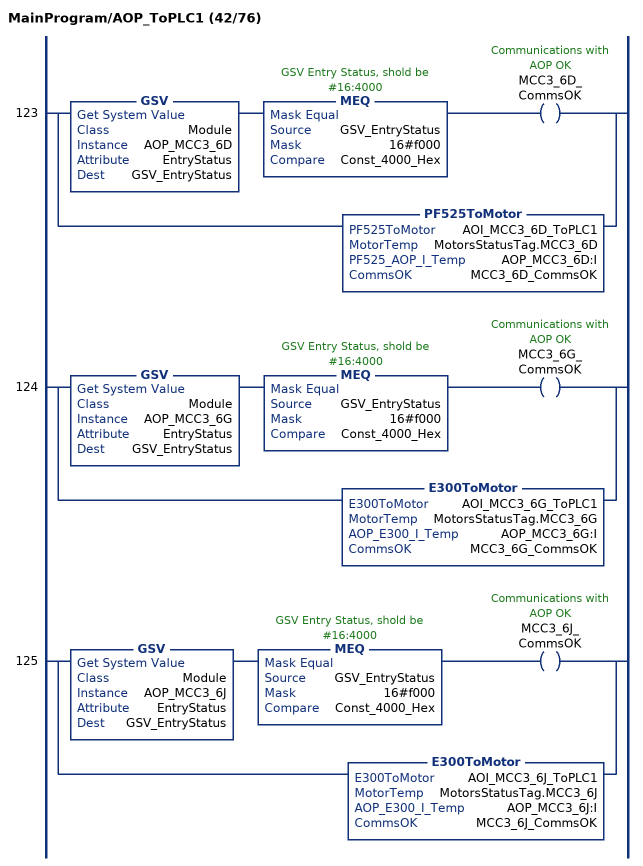
   123: [GSV(Module,AOP_MCC3_6D,EntryStatus,GSV_EntryStatus) MEQ(GSV_EntryStatus,16#f000,Const_4000_Hex) OTE(MCC3_6D_CommsOK) ,PF525ToMotor(AOI_MCC3_6D_ToPLC1,MotorsStatusTag.MCC3_6D,AOP_MCC3_6D:I,MCC3_6D_CommsOK) ];
   124: [GSV(Module,AOP_MCC3_6G,EntryStatus,GSV_EntryStatus) MEQ(GSV_EntryStatus,16#f000,Const_4000_Hex) OTE(MCC3_6G_CommsOK) ,E300ToMotor(AOI_MCC3_6G_ToPLC1,MotorsStatusTag.MCC3_6G,AOP_MCC3_6G:I,MCC3_6G_CommsOK) ];
   125: [GSV(Module,AOP_MCC3_6J,EntryStatus,GSV_EntryStatus) MEQ(GSV_EntryStatus,16#f000,Const_4000_Hex) OTE(MCC3_6J_CommsOK) ,E300ToMotor(AOI_MCC3_6J_ToPLC1,MotorsStatusTag.MCC3_6J,AOP_MCC3_6J:I,MCC3_6J_CommsOK) ];
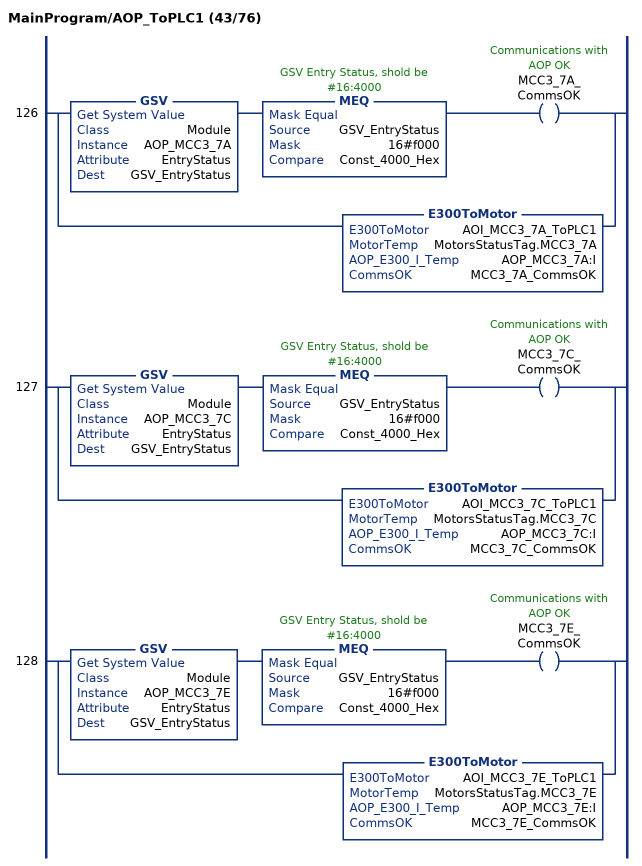
   126: [GSV(Module,AOP_MCC3_7A,EntryStatus,GSV_EntryStatus) MEQ(GSV_EntryStatus,16#f000,Const_4000_Hex) OTE(MCC3_7A_CommsOK) ,E300ToMotor(AOI_MCC3_7A_ToPLC1,MotorsStatusTag.MCC3_7A,AOP_MCC3_7A:I,MCC3_7A_CommsOK) ];
   127: [GSV(Module,AOP_MCC3_7C,EntryStatus,GSV_EntryStatus) MEQ(GSV_EntryStatus,16#f000,Const_4000_Hex) OTE(MCC3_7C_CommsOK) ,E300ToMotor(AOI_MCC3_7C_ToPLC1,MotorsStatusTag.MCC3_7C,AOP_MCC3_7C:I,MCC3_7C_CommsOK) ];
   128: [GSV(Module,AOP_MCC3_7E,EntryStatus,GSV_EntryStatus) MEQ(GSV_EntryStatus,16#f000,Const_4000_Hex) OTE(MCC3_7E_CommsOK) ,E300ToMotor(AOI_MCC3_7E_ToPLC1,MotorsStatusTag.MCC3_7E,AOP_MCC3_7E:I,MCC3_7E_CommsOK) ];
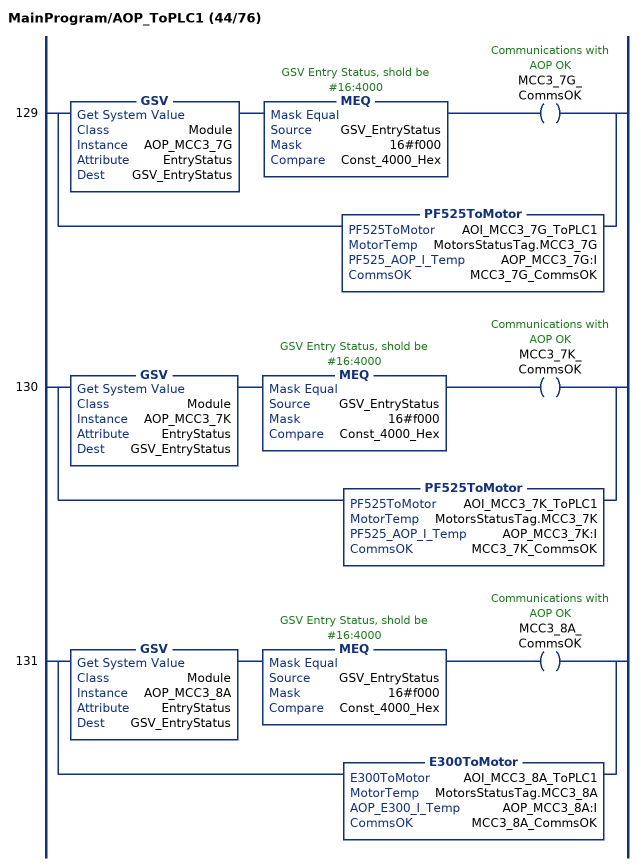
   129: [GSV(Module,AOP_MCC3_7G,EntryStatus,GSV_EntryStatus) MEQ(GSV_EntryStatus,16#f000,Const_4000_Hex) OTE(MCC3_7G_CommsOK) ,PF525ToMotor(AOI_MCC3_7G_ToPLC1,MotorsStatusTag.MCC3_7G,AOP_MCC3_7G:I,MCC3_7G_CommsOK) ];
   130: [GSV(Module,AOP_MCC3_7K,EntryStatus,GSV_EntryStatus) MEQ(GSV_EntryStatus,16#f000,Const_4000_Hex) OTE(MCC3_7K_CommsOK) ,PF525ToMotor(AOI_MCC3_7K_ToPLC1,MotorsStatusTag.MCC3_7K,AOP_MCC3_7K:I,MCC3_7K_CommsOK) ];
   131: [GSV(Module,AOP_MCC3_8A,EntryStatus,GSV_EntryStatus) MEQ(GSV_EntryStatus,16#f000,Const_4000_Hex) OTE(MCC3_8A_CommsOK) ,E300ToMotor(AOI_MCC3_8A_ToPLC1,MotorsStatusTag.MCC3_8A,AOP_MCC3_8A:I,MCC3_8A_CommsOK) ];
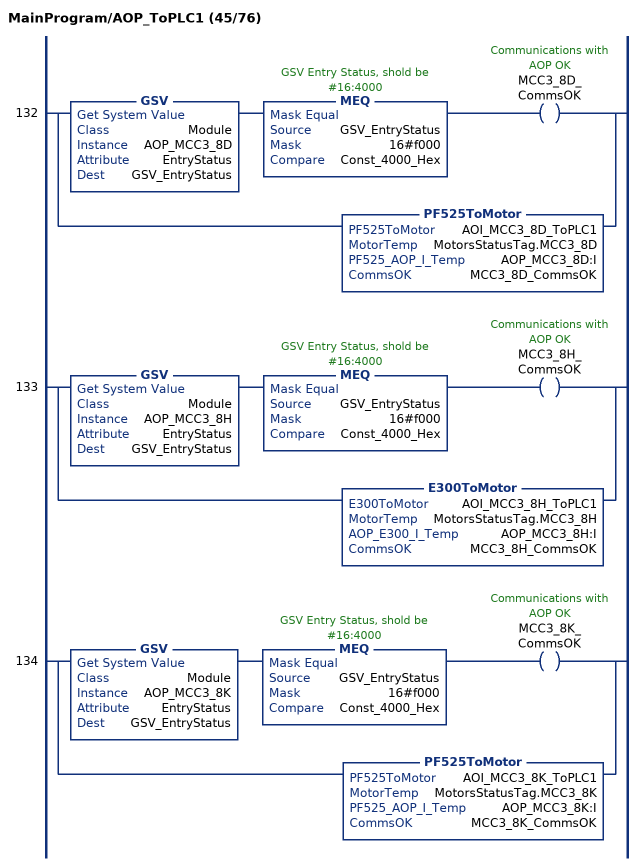
   132: [GSV(Module,AOP_MCC3_8D,EntryStatus,GSV_EntryStatus) MEQ(GSV_EntryStatus,16#f000,Const_4000_Hex) OTE(MCC3_8D_CommsOK) ,PF525ToMotor(AOI_MCC3_8D_ToPLC1,MotorsStatusTag.MCC3_8D,AOP_MCC3_8D:I,MCC3_8D_CommsOK) ];
   133: [GSV(Module,AOP_MCC3_8H,EntryStatus,GSV_EntryStatus) MEQ(GSV_EntryStatus,16#f000,Const_4000_Hex) OTE(MCC3_8H_CommsOK) ,E300ToMotor(AOI_MCC3_8H_ToPLC1,MotorsStatusTag.MCC3_8H,AOP_MCC3_8H:I,MCC3_8H_CommsOK) ];
   134: [GSV(Module,AOP_MCC3_8K,EntryStatus,GSV_EntryStatus) MEQ(GSV_EntryStatus,16#f000,Const_4000_Hex) OTE(MCC3_8K_CommsOK) ,PF525ToMotor(AOI_MCC3_8K_ToPLC1,MotorsStatusTag.MCC3_8K,AOP_MCC3_8K:I,MCC3_8K_CommsOK) ];
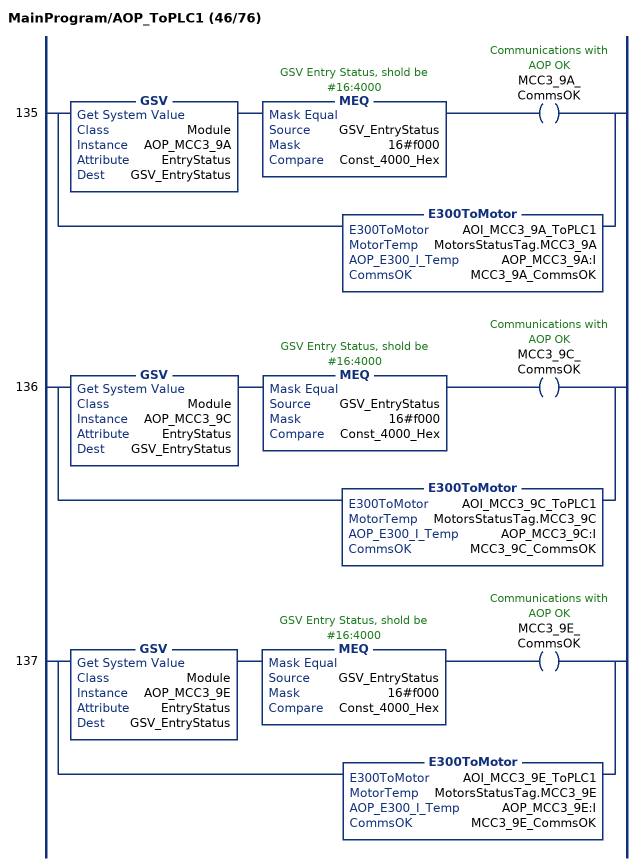
   135: [GSV(Module,AOP_MCC3_9A,EntryStatus,GSV_EntryStatus) MEQ(GSV_EntryStatus,16#f000,Const_4000_Hex) OTE(MCC3_9A_CommsOK) ,E300ToMotor(AOI_MCC3_9A_ToPLC1,MotorsStatusTag.MCC3_9A,AOP_MCC3_9A:I,MCC3_9A_CommsOK) ];
   136: [GSV(Module,AOP_MCC3_9C,EntryStatus,GSV_EntryStatus) MEQ(GSV_EntryStatus,16#f000,Const_4000_Hex) OTE(MCC3_9C_CommsOK) ,E300ToMotor(AOI_MCC3_9C_ToPLC1,MotorsStatusTag.MCC3_9C,AOP_MCC3_9C:I,MCC3_9C_CommsOK) ];
   137: [GSV(Module,AOP_MCC3_9E,EntryStatus,GSV_EntryStatus) MEQ(GSV_EntryStatus,16#f000,Const_4000_Hex) OTE(MCC3_9E_CommsOK) ,E300ToMotor(AOI_MCC3_9E_ToPLC1,MotorsStatusTag.MCC3_9E,AOP_MCC3_9E:I,MCC3_9E_CommsOK) ];
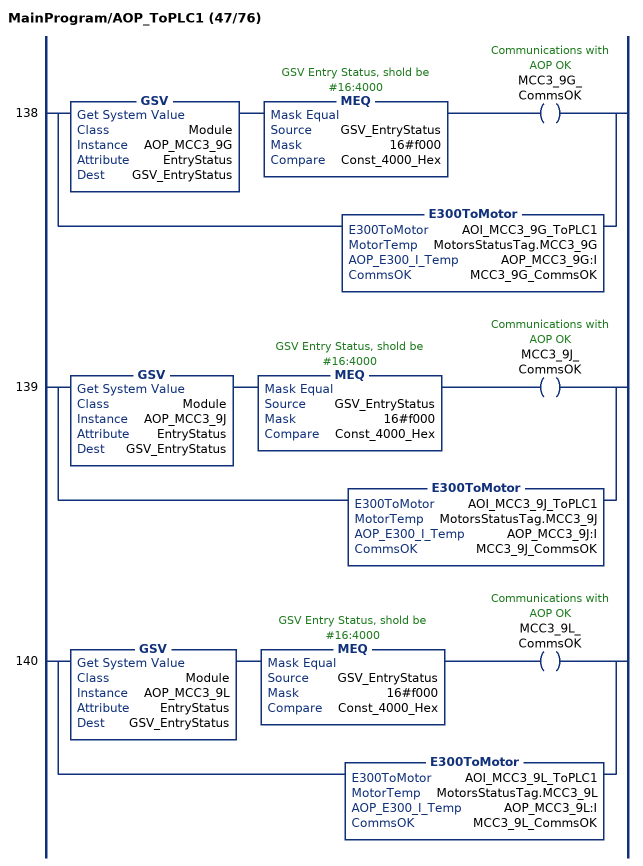
   138: [GSV(Module,AOP_MCC3_9G,EntryStatus,GSV_EntryStatus) MEQ(GSV_EntryStatus,16#f000,Const_4000_Hex) OTE(MCC3_9G_CommsOK) ,E300ToMotor(AOI_MCC3_9G_ToPLC1,MotorsStatusTag.MCC3_9G,AOP_MCC3_9G:I,MCC3_9G_CommsOK) ];
   139: [GSV(Module,AOP_MCC3_9J,EntryStatus,GSV_EntryStatus) MEQ(GSV_EntryStatus,16#f000,Const_4000_Hex) OTE(MCC3_9J_CommsOK) ,E300ToMotor(AOI_MCC3_9J_ToPLC1,MotorsStatusTag.MCC3_9J,AOP_MCC3_9J:I,MCC3_9J_CommsOK) ];
   140: [GSV(Module,AOP_MCC3_9L,EntryStatus,GSV_EntryStatus) MEQ(GSV_EntryStatus,16#f000,Const_4000_Hex) OTE(MCC3_9L_CommsOK) ,E300ToMotor(AOI_MCC3_9L_ToPLC1,MotorsStatusTag.MCC3_9L,AOP_MCC3_9L:I,MCC3_9L_CommsOK) ];
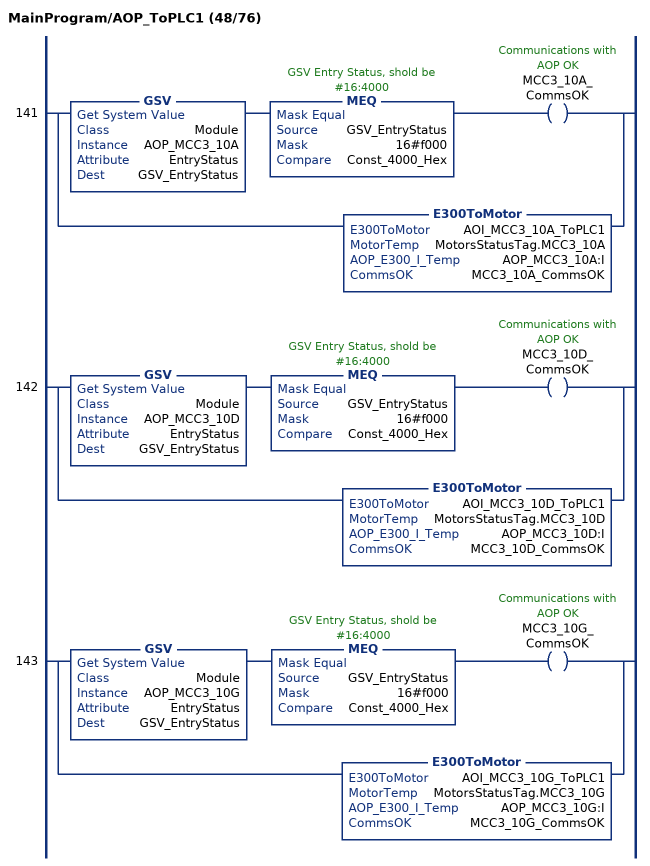
   141: [GSV(Module,AOP_MCC3_10A,EntryStatus,GSV_EntryStatus) MEQ(GSV_EntryStatus,16#f000,Const_4000_Hex) OTE(MCC3_10A_CommsOK) ,E300ToMotor(AOI_MCC3_10A_ToPLC1,MotorsStatusTag.MCC3_10A,AOP_MCC3_10A:I,MCC3_10A_CommsOK) ];
   142: [GSV(Module,AOP_MCC3_10D,EntryStatus,GSV_EntryStatus) MEQ(GSV_EntryStatus,16#f000,Const_4000_Hex) OTE(MCC3_10D_CommsOK) ,E300ToMotor(AOI_MCC3_10D_ToPLC1,MotorsStatusTag.MCC3_10D,AOP_MCC3_10D:I,MCC3_10D_CommsOK) ];
   143: [GSV(Module,AOP_MCC3_10G,EntryStatus,GSV_EntryStatus) MEQ(GSV_EntryStatus,16#f000,Const_4000_Hex) OTE(MCC3_10G_CommsOK) ,E300ToMotor(AOI_MCC3_10G_ToPLC1,MotorsStatusTag.MCC3_10G,AOP_MCC3_10G:I,MCC3_10G_CommsOK) ];
